FUNCTION_BLOCK FB_ResetSequence IMPLEMENTS I_ResetSequence
VAR

END_VAR

{warning 'Add method implementation '}
METHOD IsReset : BOOL
END_METHOD

END_FUNCTION_BLOCK

(* stored: Version 1.1.0.1
   POU FB_ResetSequence: Id {872eab31-dd48-4741-9e11-11730b82cd7c}, SpecialFunc None
   Method IsReset: Id {3d1237a0-fc42-483a-85ce-67f0844a3455} *)
